// TIA Portal V21 export
FUNCTION_BLOCK "FB_Sensores"   // FB1, LAD
TITLE = Asignacion de estados del proceso
{ S7_Optimized_Access := 'TRUE' }
// stored: MemoryReserve 100, SetENOAutomatically false
   VAR_INPUT
      High_sensor : Bool;
      Low_sensor : Bool;
      "At left" : Bool;
      "At right" : Bool;
      Reset_estados : Bool;
      Loaded : Bool;
      "At left exit" : Bool;
      "At right exit" : Bool;
   END_VAR
   VAR_OUTPUT
      Clasificando : Bool;
      "Caja Alta" : Bool;
      "Caja Baja" : Bool;
   END_VAR
   VAR_IN_OUT
      CT_Total : Int;
      CT_Cajas_Altas : Int;
      CT_Cajas_Bajas : Int;
   END_VAR
   VAR
      Mem_At_left : Bool;
      Mem_At_right : Bool;
      Mem_clasificando : Bool;
      Mem_At_left_exit : Bool;
      Mem_At_right_exit : Bool;
   END_VAR
   VAR_TEMP   // added for the SCL form of the ladder/FBD networks
      _w1 : Bool;
      _w2 : Bool;
   END_VAR
BEGIN

REGION Network 1: Estado: Clasificando
   // Inicio: Pallet llega a sensor de carga "Loaded"
   // Fin: Pallet sale de sensores de inicio laterales (At_Left/Right_Entry)
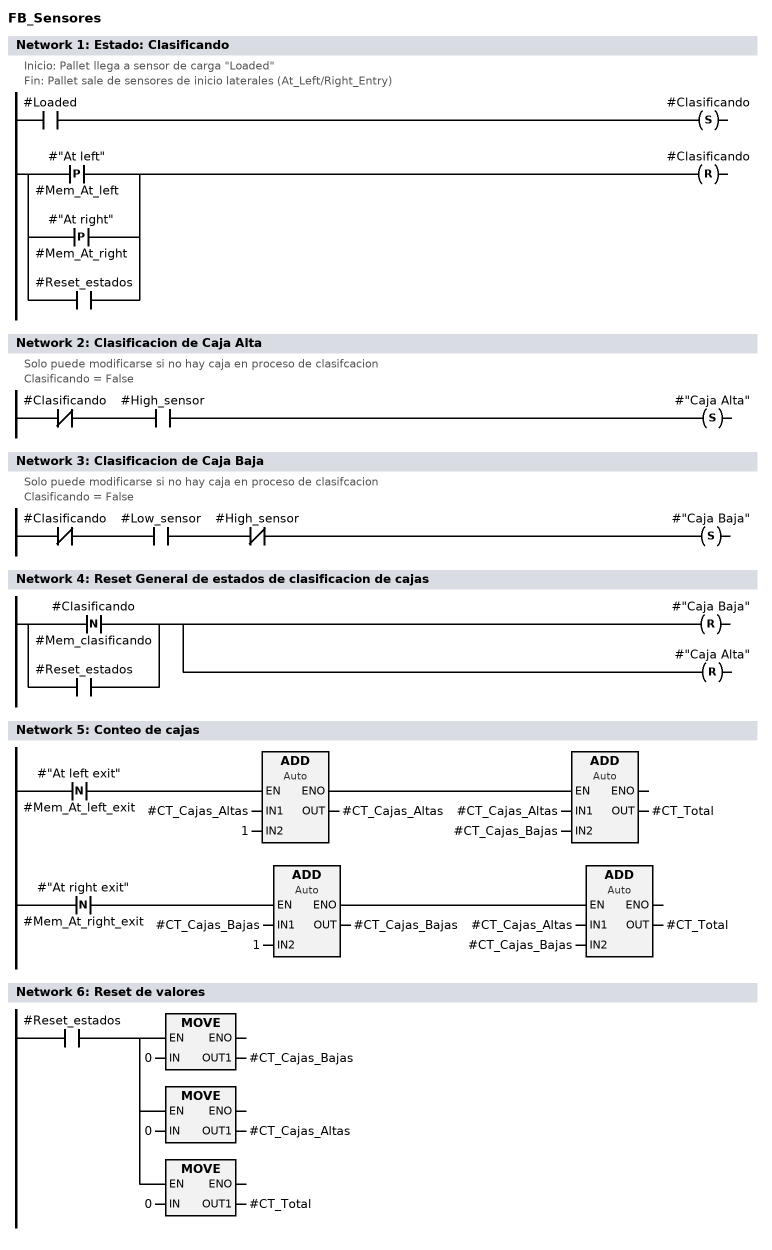
   RUNG wire#powerrail
      Contact( #Loaded )
      S_Coil( #Clasificando )
   END_RUNG
   RUNG wire#powerrail
      P_Contact(operand := #"At left", bit := #Mem_At_left)
      wire#w1
      R_Coil( #Clasificando )
   END_RUNG
   RUNG wire#powerrail
      P_Contact(operand := #"At right", bit := #Mem_At_right)
   END_RUNG wire#w1
   RUNG wire#powerrail
      Contact( #Reset_estados )
   END_RUNG wire#w1
   // the same network as SCL:
   IF #Loaded THEN #Clasificando := TRUE; END_IF;
   #_w1 := #"At left" AND NOT #Mem_At_left;   // rising edge of #"At left"
   #Mem_At_left := #"At left";
   #_w2 := #"At right" AND NOT #Mem_At_right;   // rising edge of #"At right"
   #Mem_At_right := #"At right";
   IF #_w1 OR #_w2 OR #Reset_estados THEN #Clasificando := FALSE; END_IF;
END_REGION

REGION Network 2: Clasificacion de Caja Alta
   // Solo puede modificarse si no hay caja en proceso de clasifcacion
   // Clasificando = False
   RUNG wire#powerrail
      I_Contact( #Clasificando )
      Contact( #High_sensor )
      S_Coil( #"Caja Alta" )
   END_RUNG
   // the same network as SCL:
   IF NOT #Clasificando AND #High_sensor THEN #"Caja Alta" := TRUE; END_IF;
END_REGION

REGION Network 3: Clasificacion de Caja Baja
   // Solo puede modificarse si no hay caja en proceso de clasifcacion
   // Clasificando = False
   RUNG wire#powerrail
      I_Contact( #Clasificando )
      Contact( #Low_sensor )
      I_Contact( #High_sensor )
      S_Coil( #"Caja Baja" )
   END_RUNG
   // the same network as SCL:
   IF NOT #Clasificando AND #Low_sensor AND NOT #High_sensor THEN #"Caja Baja" := TRUE; END_IF;
END_REGION

REGION Network 4: Reset General de estados de clasificacion de cajas
   RUNG wire#powerrail
      N_Contact(operand := #Clasificando, bit := #Mem_clasificando)
      wire#w1
      R_Coil( #"Caja Baja" )
   END_RUNG
   RUNG wire#powerrail
      Contact( #Reset_estados )
   END_RUNG wire#w1
   RUNG wire#w1
      R_Coil( #"Caja Alta" )
   END_RUNG
   // the same network as SCL:
   #_w1 := NOT #Clasificando AND #Mem_clasificando;   // falling edge of #Clasificando
   #Mem_clasificando := #Clasificando;
   IF #_w1 OR #Reset_estados THEN
       #"Caja Baja" := FALSE;
       #"Caja Alta" := FALSE;
   END_IF;
END_REGION

REGION Network 5: Conteo de cajas
   RUNG wire#powerrail
      N_Contact(operand := #"At left exit", bit := #Mem_At_left_exit)
      Add(in1 := #CT_Cajas_Altas, in2 := 1, out => #CT_Cajas_Altas)
      Add(in1 := #CT_Cajas_Altas, in2 := #CT_Cajas_Bajas, out => #CT_Total)
   END_RUNG
   RUNG wire#powerrail
      N_Contact(operand := #"At right exit", bit := #Mem_At_right_exit)
      Add(in1 := #CT_Cajas_Bajas, in2 := 1, out => #CT_Cajas_Bajas)
      Add(in1 := #CT_Cajas_Altas, in2 := #CT_Cajas_Bajas, out => #CT_Total)
   END_RUNG
   // the same network as SCL:
   #_w1 := NOT #"At left exit" AND #Mem_At_left_exit;   // falling edge of #"At left exit"
   #Mem_At_left_exit := #"At left exit";
   IF #_w1 THEN
       #CT_Cajas_Altas := #CT_Cajas_Altas + 1;
       #CT_Total := #CT_Cajas_Altas + #CT_Cajas_Bajas;
   END_IF;
   #_w2 := NOT #"At right exit" AND #Mem_At_right_exit;   // falling edge of #"At right exit"
   #Mem_At_right_exit := #"At right exit";
   IF #_w2 THEN
       #CT_Cajas_Bajas := #CT_Cajas_Bajas + 1;
       #CT_Total := #CT_Cajas_Altas + #CT_Cajas_Bajas;
   END_IF;
END_REGION

REGION Network 6: Reset de valores
   RUNG wire#powerrail
      Contact( #Reset_estados )
      wire#w1
      Move(in := 0, out1 => #CT_Cajas_Bajas)
   END_RUNG
   RUNG wire#w1
      Move(in := 0, out1 => #CT_Cajas_Altas)
   END_RUNG
   RUNG wire#w1
      Move(in := 0, out1 => #CT_Total)
   END_RUNG
   // the same network as SCL:
   IF #Reset_estados THEN
       #CT_Cajas_Bajas := 0;
       #CT_Cajas_Altas := 0;
       #CT_Total := 0;
   END_IF;
END_REGION
END_FUNCTION_BLOCK
